Fanuc TP program (LS listing): TOOL01_SOUFFLAGE_OFF.LS

/PROG  TOOL01_SOUFFLAGE_OFF
/ATTR
OWNER		= MNEDITOR;
COMMENT		= "Soufflage OFF";
PROG_SIZE	= 194;
CREATE		= DATE 25-04-30  TIME 08:27:44;
MODIFIED	= DATE 25-04-30  TIME 08:27:44;
FILE_NAME	= TOOL01_S;
VERSION		= 0;
LINE_COUNT	= 0;
MEMORY_SIZE	= 438;
PROTECT		= READ_WRITE;
TCD:  STACK_SIZE	= 0,
      TASK_PRIORITY	= 50,
      TIME_SLICE	= 0,
      BUSY_LAMP_OFF	= 0,
      ABORT_REQUEST	= 0,
      PAUSE_REQUEST	= 0;
DEFAULT_GROUP	= 1,*,*,*,*;
CONTROL_CODE	= 00000000 00000000;
/APPL
/MN
/POS
/END
